(* Logix 5000 project; controller EuniceF_Lab1 vendor 1 type 14 code 150 rev 37.11; software revision 37.00 *)

TASK MainTask (continuous, watchdog 500 ms) : MainProgram

MODULES
   Local : vendor 1 type 14 code 150 (Compact 0, rev 37.11)
      Discrete_IO : Embedded (Compact 1, rev 3.1, Output RPI 20 ms)
      Analog_IO : Embedded (Compact 2, rev 1.1, Output RPI 80 ms)
      Counters : Embedded (Compact 3, rev 1.1, Output RPI 20 ms)
END_MODULES

VAR_GLOBAL   (* controller tags *)
   C1 : COUNTER := (PRE := 2);
   CloseTime : STRING;
   Cmess : STRING := ' Press Done DI15 ';
   ContinueMess : STRING := ' K-factor,';
   Countfor60cm : DINT;
   CurrConst : STRING := ' Filling Level: ';
   CurrHeight : DINT;
   CurrHeightS : STRING;
   CurrHMess : STRING;
   CurrHUnit : STRING;
   Defalut_Kfactor : DINT := 13403;
   DelayTime : TIMER := (PRE := 60000);
   Diif_Pressure : ALIAS FOR Local:2:I.Ch3Data;
   Done : ALIAS FOR Local:1:I.Data.15;
   Drain_Manual : ALIAS FOR Local:1:I.Data.4;
   DrainClose : DINT;
   DrainEnd : STRING := 'Drain ends in:';
   DrainHeight : DINT;
   DrainInterMess : STRING;
   DrainTime : DINT;
   DrainTimeS : STRING;
   DrainValve : ALIAS FOR Local:1:O.Data.10;
   DUMPB : ALIAS FOR Local:1:I.Data.5;
   Emerg_Resume : STRING := 'Press DI04 to Drain';
   Emerg_State : STRING := 'Emergency stop Pressed  ';
   Fill_Valve : ALIAS FOR Local:2:O.Ch1Data;
   Full : INT := 29208;
   Full_Btn : ALIAS FOR Local:1:I.Data.13;
   Good : ALIAS FOR Local:1:I.Data.14;
   Half : INT := -288;
   Half_Btn : ALIAS FOR Local:1:I.Data.12;
   Height : REAL;
   HSC1_CurentCount : ALIAS FOR Local:3:I.Ctr0CurrentCount;
   HSCMessage : STRING;
   InterMess : STRING;
   K_factor : DINT;
   KfactorMessage : STRING;
   lastrunInter : STRING;
   LevelMax : DINT := 16923;
   LevelMess : STRING;
   LevelMin : DINT := -27413;
   LevelUnit : STRING := ' cm';
   MainMessage : STRING;
   mess : STRING := ' to continue';
   Mixer : ALIAS FOR Local:1:O.Data.9;
   Mixer1 : ALIAS FOR Local:1:O.Data.9;
   MixTime : DINT;
   MixTimeLeft : DINT;
   MixTimeLeftMess : STRING;
   MixTimeMess : STRING := 'The Mixer will stop in: ';
   PressInterMess : STRING;
   PressionMess : STRING;
   PressMess : STRING := 'Draining level: ';
   PressS : STRING;
   PressUnit : STRING := 'EU';
   price : DINT;
   PRICEInter : STRING;
   priceMess : STRING := ' The price is : ';
   pricemess2 : STRING;
   priceS : STRING;
   priceUnit : STRING := ' dollars ';
   Prove : ALIAS FOR Local:1:I.Data.7;
   provebMessage : STRING := 'Press DI07';
   ProveMess : STRING := ' prove to start';
   Pump : ALIAS FOR Local:1:O.Data.8;
   PumpButton : STRING := ': Press DI14 when you reach 60 cm';
   PumpMessage : STRING := ' Pump on, Press DI14 when you reach';
   Quarter : INT := -15037;
   Quarter_Btn : ALIAS FOR Local:1:I.Data.11;
   Reset_HSC : ALIAS FOR Local:3:O.Ctr0SoftPreset;
   Round : DINT;
   SEQ : DINT;
   Start : ALIAS FOR Local:1:I.Data.1;
   Start1 : ALIAS FOR Local:1:I.Data.11;
   Start2 : ALIAS FOR Local:1:I.Data.12;
   StartButton : STRING := ' to start ';
   StartMessage : STRING := 'Press DI01';
   Status : STRING;
   Stop : ALIAS FOR Local:1:I.Data.2;
   Stop_Emergency : STRING := 'Press DI02 ';
   Stop_MainMessage : STRING;
   Stopbutton : STRING := ' for the emergency stop';
   StopPressed : STRING;
   T1 : TIMER := (PRE := 10000);
   T3 : TIMER := (PRE := 10000);
   T8 : TIMER := (PRE := 12000);
   TargetTicks : DINT;
   Time : TIMER := (PRE := 10000);
   TimerDrain : DINT;
   V1 : DINT;
   V2 : DINT;
   Value : ALIAS FOR Local:2:I.Ch0Data;
   Valve_Position : ALIAS FOR Local:2:O.Ch1Data;
   valveMess : STRING := ' to open';
   ValveTime : STRING := 'The valve will close in: ';
   Vol_Unit : STRING := 'ml';
   VolInter : STRING;
   VolString : STRING;
   Volume : DINT;
   VolumeMess : STRING;
   VolumeStatus : STRING := ' Volume: ';
   Zero : ALIAS FOR Local:1:I.Data.3;
END_VAR

PROGRAM MainProgram   (* main routine MainRoutine *)
VAR
   dump : BOOL;
   lastTurn : DINT;
   TimeDrain : TIMER := (PRE := 120000);
   TimeEndDrain : TIMER := (PRE := 60000);
   V3 : DINT;
END_VAR

ROUTINE MainRoutine   (* ladder *)
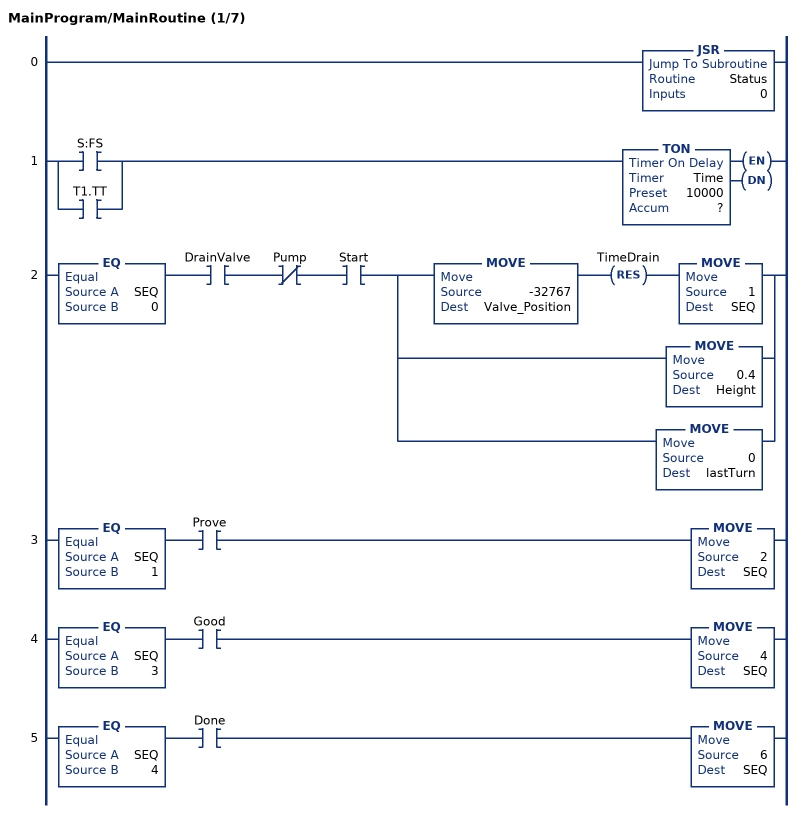
   0: JSR(Status,0);
   1: [XIC(S:FS) ,XIC(T1.TT) ]TON(Time,?,?);
   2: EQ(SEQ,0)XIC(DrainValve)XIO(Pump)XIC(Start)[MOVE(-32767,Valve_Position) RES(TimeDrain) MOVE(1,SEQ) ,MOVE(0.4,Height) ,MOVE(0,lastTurn) ];
   3: EQ(SEQ,1)XIC(Prove)MOVE(2,SEQ);
   4: EQ(SEQ,3)XIC(Good)MOVE(4,SEQ);
   5: EQ(SEQ,4)XIC(Done)MOVE(6,SEQ);
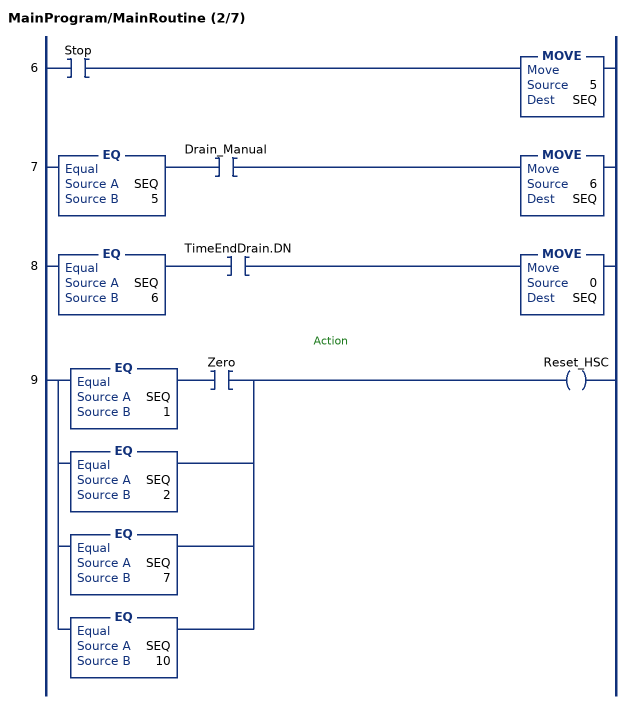
   6: XIC(Stop)MOVE(5,SEQ);
   7: EQ(SEQ,5)XIC(Drain_Manual)MOVE(6,SEQ);
   8: EQ(SEQ,6)XIC(TimeEndDrain.DN)MOVE(0,SEQ);
   // Action
   9: [EQ(SEQ,1) XIC(Zero) ,EQ(SEQ,2) ,EQ(SEQ,7) ,EQ(SEQ,10) ]OTE(Reset_HSC);
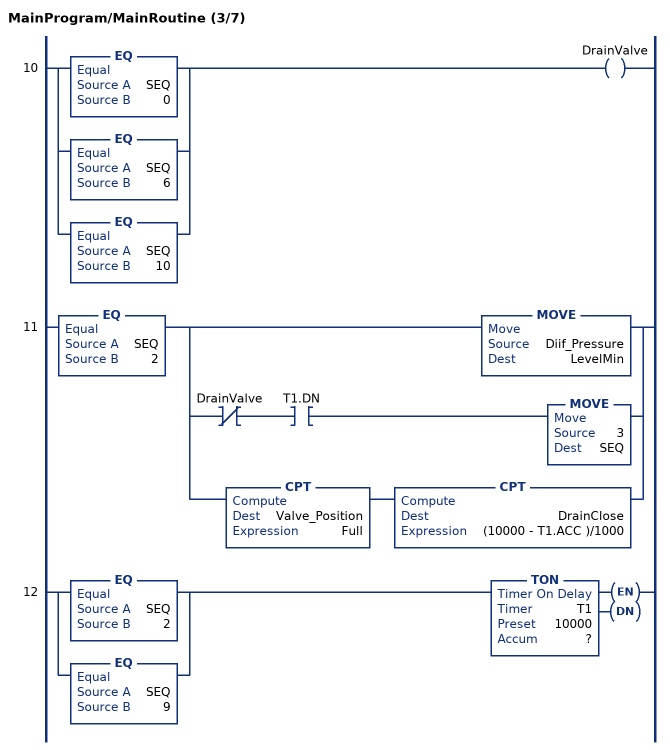
   10: [EQ(SEQ,0) ,EQ(SEQ,6) ,EQ(SEQ,10) ]OTE(DrainValve);
   11: EQ(SEQ,2)[MOVE(Diif_Pressure,LevelMin) ,XIO(DrainValve) XIC(T1.DN) MOVE(3,SEQ) ,CPT(Valve_Position,Full) CPT(DrainClose,(10000 - T1.ACC )/1000) ];
   12: [EQ(SEQ,2) ,EQ(SEQ,9) ]TON(T1,?,?);
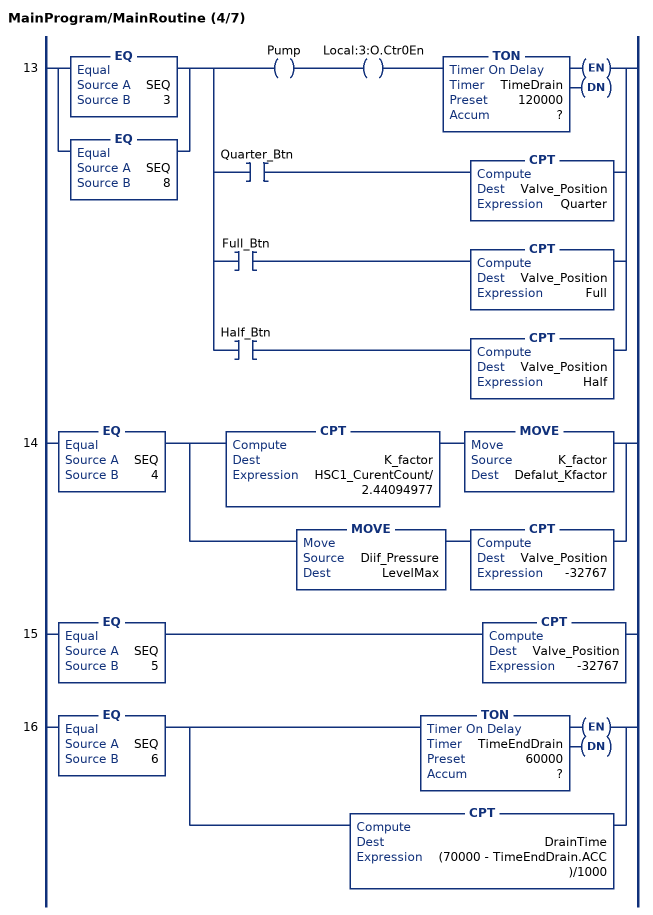
   13: [EQ(SEQ,3) ,EQ(SEQ,8) ][OTE(Pump) OTE(Local:3:O.Ctr0En) TON(TimeDrain,?,?) ,XIC(Quarter_Btn) CPT(Valve_Position,Quarter) ,XIC(Full_Btn) CPT(Valve_Position,Full) ,XIC(Half_Btn) CPT(Valve_Position,Half) ];
   14: EQ(SEQ,4)[CPT(K_factor,HSC1_CurentCount/ 2.44094977) MOVE(K_factor,Defalut_Kfactor) ,MOVE(Diif_Pressure,LevelMax) CPT(Valve_Position,-32767) ];
   15: EQ(SEQ,5)CPT(Valve_Position,-32767);
   16: EQ(SEQ,6)[TON(TimeEndDrain,?,?) ,CPT(DrainTime,(70000 - TimeEndDrain.ACC )/1000) ];
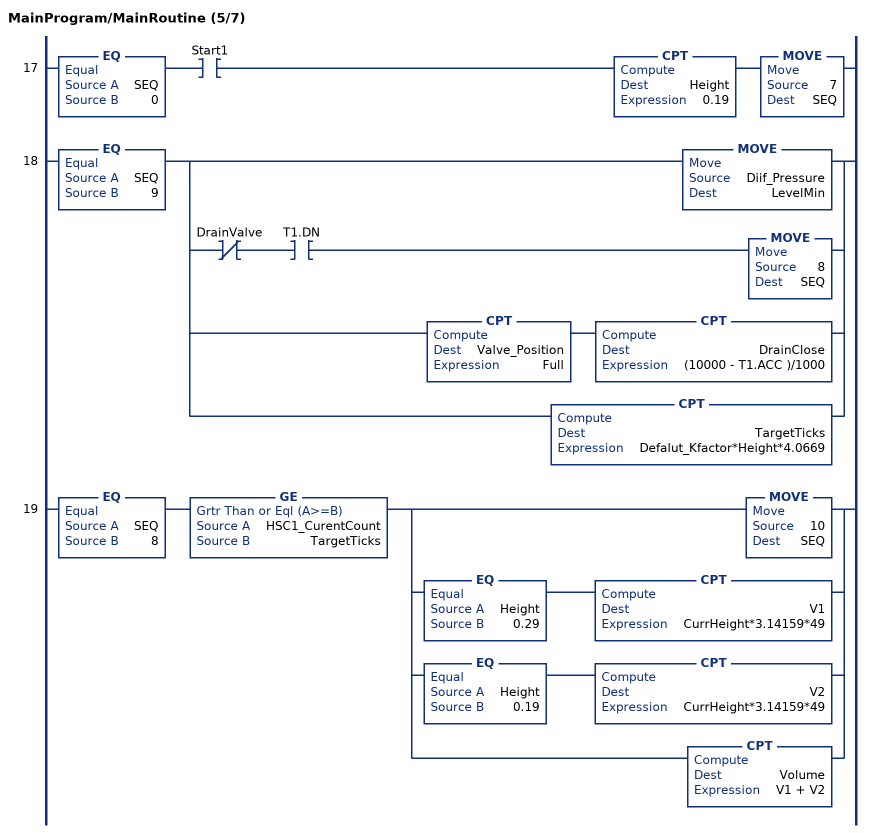
   17: EQ(SEQ,0)XIC(Start1)CPT(Height,0.19)MOVE(7,SEQ);
   18: EQ(SEQ,9)[MOVE(Diif_Pressure,LevelMin) ,XIO(DrainValve) XIC(T1.DN) MOVE(8,SEQ) ,CPT(Valve_Position,Full) CPT(DrainClose,(10000 - T1.ACC )/1000) ,CPT(TargetTicks,Defalut_Kfactor*Height*4.0669) ];
   19: EQ(SEQ,8)GE(HSC1_CurentCount,TargetTicks)[MOVE(10,SEQ) ,EQ(Height,0.29) CPT(V1,CurrHeight*3.14159*49) ,EQ(Height,0.19) CPT(V2,CurrHeight*3.14159*49) ,CPT(Volume,V1 + V2) ];
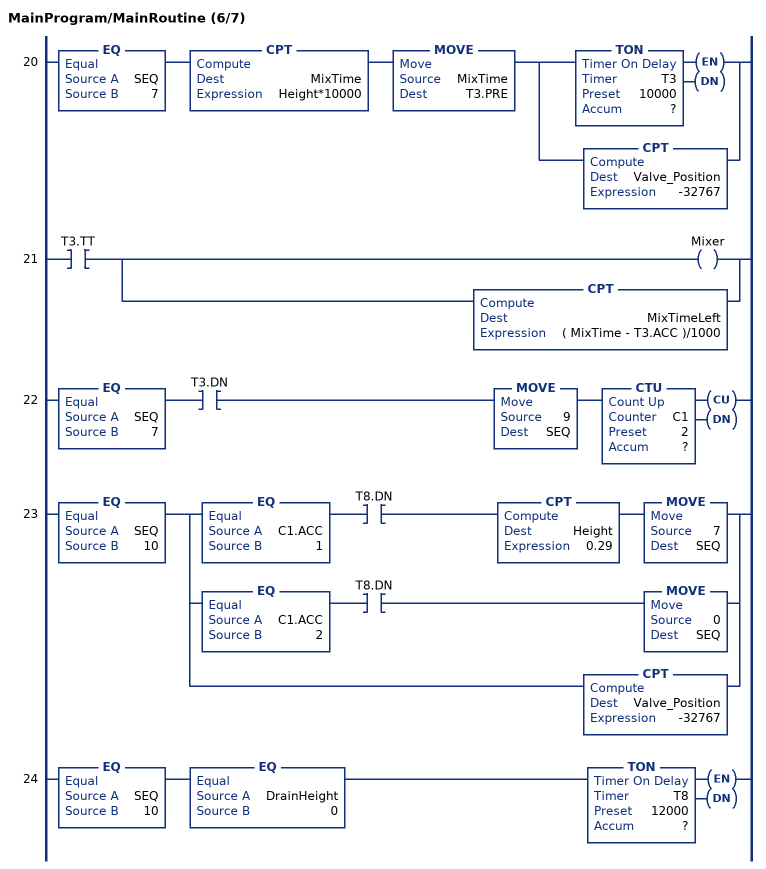
   20: EQ(SEQ,7)CPT(MixTime,Height*10000)MOVE(MixTime,T3.PRE)[TON(T3,?,?) ,CPT(Valve_Position,-32767) ];
   21: XIC(T3.TT)[OTE(Mixer) ,CPT(MixTimeLeft,( MixTime - T3.ACC )/1000) ];
   22: EQ(SEQ,7)XIC(T3.DN)MOVE(9,SEQ)CTU(C1,?,?);
   23: EQ(SEQ,10)[EQ(C1.ACC,1) XIC(T8.DN) CPT(Height,0.29) MOVE(7,SEQ) ,EQ(C1.ACC,2) XIC(T8.DN) MOVE(0,SEQ) ,CPT(Valve_Position,-32767) ];
   24: EQ(SEQ,10)EQ(DrainHeight,0)TON(T8,?,?);
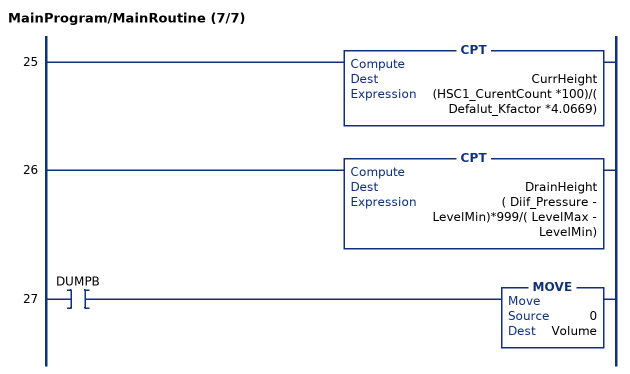
   25: CPT(CurrHeight,(HSC1_CurentCount *100)/( Defalut_Kfactor *4.0669));
   26: CPT(DrainHeight,( Diif_Pressure - LevelMin)*999/( LevelMax - LevelMin));
   27: XIC(DUMPB)MOVE(0,Volume);
END_ROUTINE

ROUTINE Status   (* structured text *)
   if SEQ=0 then
   	concat(StartMessage,StartButton,MainMessage);
   end_if;
   
   //Waiting
   if SEQ=1 then
   	concat(provebMessage,ProveMess,MainMessage);
   	concat(Stop_Emergency,Stopbutton,Stop_MainMessage);
   end_if;
   
   //Closing valve
   if SEQ=2 or SEQ=9 then
   	DTOS(DrainClose,CloseTime);
   	concat(ValveTime,CloseTime,MainMessage);
   	concat(Stop_Emergency,Stopbutton,Stop_MainMessage);
   end_if;
   
   //The valve is pumping
   if SEQ=3 then
   	DTOS(HSC1_CurentCount,HSCMessage);
   	concat(HSCMessage,PumpButton,MainMessage);
   	concat(Stop_Emergency,Stopbutton,Stop_MainMessage);
   end_if;
   
   //Calculating and Done can be pressed
   if SEQ=4 then
   	DTOS(K_factor,KfactorMessage);
   	concat(KfactorMessage,ContinueMess,MainMessage);
   	concat(Cmess,mess,Stop_MainMessage);
   end_if;
   
   //Emergency stop has been pressed
   if SEQ=5 then
   	concat(Emerg_State,Emerg_Resume,MainMessage);
   	concat(Stop_Emergency,Stopbutton,Stop_MainMessage);
   end_if;
   
   //Drain time (after the Drain button has been pressed or the Done button has been pressed)
   if SEQ=6 or SEQ=10 then
   	DTOS(DrainTime,DrainTimeS);
   	DTOS(DrainHeight,PressS);
   	concat(PressMess,PressS,PressInterMess);
   	concat(PressInterMess,PressUnit,PressionMess);
   	concat(DrainEnd,DrainTimeS,DrainInterMess);
   	concat(PressionMess,DrainInterMess,MainMessage);
   	concat(Stop_Emergency,Stopbutton,Stop_MainMessage);
   end_if;
   
   if SEQ=8 and lastTurn = 0 then
   	DTOS(CurrHeight,CurrHeightS);
   	concat(CurrConst,CurrHeightS,CurrHMess);
   	concat(CurrHMess,LevelUnit,MainMessage);
   	concat(Stop_Emergency,Stopbutton,Stop_MainMessage);
   end_if;
   
   if SEQ=7 then
   	DTOS(MixTimeLeft,MixTimeLeftMess);
   	concat(MixTimeMess,MixTimeLeftMess,MainMessage);
   	concat(Stop_Emergency,Stopbutton,Stop_MainMessage);
   end_if;
   
   
   
   
   
   
END_ROUTINE
END_PROGRAM
